FUNCTION_BLOCK SBCalibrator (* Sonnenbatterie calibrator. Sets the battery's control mode to automatic for calibration while fully charged. *)
  (* Standard: 61499-2; Description: Requires the http communication layer. *)
  (* Version 1.0, 2017-08-27, Marc Jakobi, HTW Berlin *)
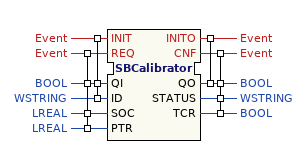
  EVENT_INPUT
    INIT WITH QI, ID; (* Initialization Event *)
    REQ WITH SOC, QI, PTR; (* Normal Execution Request *)
  END_EVENT
  EVENT_OUTPUT
    INITO WITH QO; (* Initialization confirm *)
    CNF WITH QO, STATUS, TCR; (* Execution Confirmation *)
  END_EVENT
  VAR_INPUT
    QI : BOOL; (* Input event qualifier *)
    ID : WSTRING; (* Connection identifier (ip:port) *)
    SOC : LREAL; (* State of charge [0,..,1] *)
    PTR : LREAL; (* Power used to release from trickle charge in W *)
  END_VAR
  VAR_OUTPUT
    QO : BOOL; (* Output event qualifier *)
    STATUS : WSTRING; (* HTTP responses *)
    TCR : BOOL; (* true, if battery has just been released from trickle charge *)
  END_VAR
  FBS
    FullyCharged : F_GE(IN2 := LREAL#1);
    TrickleCharge : F_EQ(IN2 := UINT#42);
    NonAuto : F_GE(IN2 := UINT#20);
    F_AND : F_AND;
    Auto2 : CLIENT_1(QI := TRUE, SD_1 := UINT#10);
    NotFull : F_LT(IN2 := LREAL#0.95);
    AutoActive : F_LT(IN2 := UINT#20);
    F_GT : F_GT(IN2 := UINT#30);
    F_OR : F_OR;
    F_AND_1 : F_AND;
    BOOL2BOOL : BOOL2BOOL;
    E_SWITCH : E_SWITCH;
    E_SWITCH_1 : E_SWITCH;
    E_SWITCH_2 : E_SWITCH;
    Auto1 : CLIENT_1(QI := TRUE, SD_1 := UINT#10);
    E_DELAY : E_DELAY(DT := T#2s);
    Manual1 : CLIENT_1(QI := TRUE, SD_1 := UINT#55);
    F_CONCAT : F_CONCAT(IN1 := WSTRING#http[);
    F_CONCAT_1 : F_CONCAT(IN2 := WSTRING#/rest/devices/battery/);
    WSTRING2WSTRING : WSTRING2WSTRING;
    Write_mode_ID : F_CONCAT(IN2 := WSTRING#C06]);
    WSTRING2WSTRING_1 : WSTRING2WSTRING;
    Write_charge_ID : F_CONCAT(IN2 := WSTRING#C24]);
    WSTRING2WSTRING_2 : WSTRING2WSTRING;
    WSTRING2WSTRING_3 : WSTRING2WSTRING;
    Manual2 : CLIENT_1(QI := TRUE, SD_1 := UINT#55);
    Charge : CLIENT_1(QI := TRUE);
    E_DELAY_1 : E_DELAY(DT := T#10s);
    E_DELAY_2 : E_DELAY(DT := T#20s);
    E_DELAY_3 : E_DELAY(DT := T#10s);
    TrickleChargeRelease : E_TF;
    E_MERGE : E_MERGE;
    UINT2UINT : UINT2UINT;
    BatteryMode : CLIENT_0_1;
    Read_mode_ID : F_CONCAT(IN2 := WSTRING#M06]);
    WSTRING2WSTRING_12 : WSTRING2WSTRING;
    F_AND_2 : F_AND;
    F_OR_1 : F_OR;
    BOOL2BOOL_2 : BOOL2BOOL;
    F_AND_3 : F_AND;
    BOOL2BOOL_3 : BOOL2BOOL;
    F_OR_2 : F_OR;
    BOOL2BOOL_1 : BOOL2BOOL;
    FB_SEL_WSTRING : FB_SEL_WSTRING(IN0 := WSTRING#SBCALIBRATOR_ERROR, IN1 := WSTRING#OK);
    BOOL2BOOL_4 : BOOL2BOOL;
    F_AND_4 : F_AND;
    E_TF : E_TF;
    BOOL2BOOL_5 : BOOL2BOOL;
    F_OR_3 : F_OR;
  END_FBS
  EVENT_CONNECTIONS
    F_OR.CNF TO BOOL2BOOL.REQ;
    BOOL2BOOL.CNF TO F_AND_1.REQ;
    FullyCharged.CNF TO NonAuto.REQ;
    NonAuto.CNF TO F_AND.REQ;
    F_AND.CNF TO E_SWITCH.EI;
    TrickleCharge.CNF TO E_SWITCH_1.EI;
    F_AND_1.CNF TO E_SWITCH_2.EI;
    E_SWITCH_2.EO0 TO FullyCharged.REQ;
    E_DELAY.EO TO Manual1.REQ;
    F_CONCAT.CNF TO WSTRING2WSTRING.REQ;
    WSTRING2WSTRING.CNF TO F_CONCAT_1.REQ;
    F_CONCAT_1.CNF TO WSTRING2WSTRING_1.REQ;
    WSTRING2WSTRING_1.CNF TO Write_mode_ID.REQ;
    Write_mode_ID.CNF TO WSTRING2WSTRING_2.REQ;
    E_SWITCH.EO0 TO TrickleCharge.REQ;
    Write_charge_ID.CNF TO WSTRING2WSTRING_3.REQ;
    E_SWITCH.EO1 TO Auto2.REQ;
    E_DELAY_1.EO TO Charge.REQ;
    E_DELAY_3.EO TO E_MERGE.EI1;
    INIT TO F_CONCAT.REQ;
    REQ TO BatteryMode.REQ;
    BatteryMode.CNF TO UINT2UINT.REQ;
    WSTRING2WSTRING_2.CNF TO Read_mode_ID.REQ;
    Read_mode_ID.CNF TO WSTRING2WSTRING_12.REQ;
    UINT2UINT.CNF TO NotFull.REQ;
    WSTRING2WSTRING_12.CNF TO BatteryMode.INIT;
    NotFull.CNF TO AutoActive.REQ;
    AutoActive.CNF TO F_GT.REQ;
    F_GT.CNF TO F_OR.REQ;
    E_SWITCH_2.EO1 TO Auto1.REQ;
    Auto1.CNF TO E_DELAY.START;
    E_SWITCH_1.EO1 TO Manual2.REQ;
    Manual2.CNF TO E_DELAY_1.START;
    BatteryMode.INITO TO Auto1.INIT;
    Auto1.INITO TO Manual1.INIT;
    Auto2.INITO TO Manual2.INIT;
    Manual1.INITO TO Write_charge_ID.REQ;
    WSTRING2WSTRING_3.CNF TO Auto2.INIT;
    Manual2.INITO TO Charge.INIT;
    Charge.INITO TO INITO;
    Manual1.CNF TO F_AND_2.REQ;
    F_OR_1.CNF TO BOOL2BOOL_2.REQ;
    Charge.CNF TO F_AND_3.REQ;
    F_AND_3.CNF TO BOOL2BOOL_3.REQ;
    F_AND_2.CNF TO BOOL2BOOL_1.REQ;
    BOOL2BOOL_1.CNF TO E_DELAY_3.START;
    F_OR_2.CNF TO BOOL2BOOL_4.REQ;
    BOOL2BOOL_4.CNF TO F_AND_4.REQ;
    BOOL2BOOL_3.CNF TO E_DELAY_2.START;
    E_DELAY_2.EO TO TrickleChargeRelease.TRUE;
    FB_SEL_WSTRING.CNF TO CNF;
    E_SWITCH_1.EO0 TO E_TF.TRUE;
    E_MERGE.EO TO E_TF.FALSE;
    E_TF.EO TO TrickleChargeRelease.FALSE;
    F_OR_3.CNF TO FB_SEL_WSTRING.REQ;
    BOOL2BOOL_5.CNF TO F_OR_3.REQ;
    F_AND_4.CNF TO BOOL2BOOL_5.REQ;
    Auto2.CNF TO E_MERGE.EI2;
    TrickleChargeRelease.EO TO F_OR_1.REQ;
    BOOL2BOOL_2.CNF TO F_OR_2.REQ;
  END_CONNECTIONS
  DATA_CONNECTIONS
    SOC TO FullyCharged.IN1;
    FullyCharged.OUT TO F_AND.IN1;
    NonAuto.OUT TO F_AND.IN2;
    SOC TO NotFull.IN1;
    F_GT.OUT TO F_OR.IN2;
    NotFull.OUT TO F_AND_1.IN1;
    F_OR.OUT TO BOOL2BOOL.IN;
    BOOL2BOOL.OUT TO F_AND_1.IN2;
    F_AND.OUT TO E_SWITCH.G;
    TrickleCharge.OUT TO E_SWITCH_1.G;
    F_AND_1.OUT TO E_SWITCH_2.G;
    ID TO F_CONCAT.IN2;
    F_CONCAT.OUT TO WSTRING2WSTRING.IN;
    WSTRING2WSTRING.OUT TO F_CONCAT_1.IN1;
    F_CONCAT_1.OUT TO WSTRING2WSTRING_1.IN;
    WSTRING2WSTRING_1.OUT TO Write_mode_ID.IN1;
    WSTRING2WSTRING_1.OUT TO Write_charge_ID.IN1;
    Write_mode_ID.OUT TO WSTRING2WSTRING_2.IN;
    Write_charge_ID.OUT TO WSTRING2WSTRING_3.IN;
    WSTRING2WSTRING_3.OUT TO Charge.ID;
    PTR TO Charge.SD_1;
    TrickleChargeRelease.Q TO TCR;
    BatteryMode.RD_1 TO UINT2UINT.IN;
    WSTRING2WSTRING_1.OUT TO Read_mode_ID.IN1;
    Read_mode_ID.OUT TO WSTRING2WSTRING_12.IN;
    WSTRING2WSTRING_12.OUT TO BatteryMode.ID;
    UINT2UINT.OUT TO F_GT.IN1;
    UINT2UINT.OUT TO NonAuto.IN1;
    UINT2UINT.OUT TO TrickleCharge.IN1;
    UINT2UINT.OUT TO AutoActive.IN1;
    AutoActive.OUT TO F_OR.IN1;
    WSTRING2WSTRING_2.OUT TO Auto2.ID;
    WSTRING2WSTRING_2.OUT TO Manual1.ID;
    WSTRING2WSTRING_2.OUT TO Auto1.ID;
    WSTRING2WSTRING_2.OUT TO Manual2.ID;
    QI TO BatteryMode.QI;
    Manual1.QO TO F_AND_2.IN1;
    Auto1.QO TO F_AND_2.IN2;
    Auto2.QO TO F_OR_1.IN2;
    F_OR_1.OUT TO BOOL2BOOL_2.IN;
    Manual2.QO TO F_AND_3.IN1;
    Charge.QO TO F_AND_3.IN2;
    F_AND_3.OUT TO BOOL2BOOL_3.IN;
    F_AND_2.OUT TO BOOL2BOOL_1.IN;
    BOOL2BOOL_1.OUT TO F_OR_1.IN1;
    BOOL2BOOL_3.OUT TO F_OR_2.IN2;
    BOOL2BOOL_2.OUT TO F_OR_2.IN1;
    FB_SEL_WSTRING.OUT TO STATUS;
    F_OR_2.OUT TO BOOL2BOOL_4.IN;
    BOOL2BOOL_4.OUT TO F_AND_4.IN2;
    BatteryMode.QO TO F_AND_4.IN1;
    F_OR_3.OUT TO FB_SEL_WSTRING.QI;
    F_OR_3.OUT TO QO;
    BOOL2BOOL_5.OUT TO F_OR_3.IN2;
    F_AND_4.OUT TO BOOL2BOOL_5.IN;
    E_TF.Q TO F_OR_3.IN1;
  END_CONNECTIONS
END_FUNCTION_BLOCK
